(* IEC 61131-3 sources: eCockpitGit/test_project/src/%F%03 Module/%POU%FB_Module/%F%SYS Values/%PRO%SYS_valueUnsigned64, 2 files *)

(* ---- %GETSET%Get.st ---- *)
VAR
END_VAR

(*%!%__DELIMITER__%!%*)
CASE SYS_valueType OF
	EValueType.digital:		SYS_valueUnsigned64	:=		TO_LWORD(SYS_valueDigital);
	EValueType.float32:		SYS_valueUnsigned64	:=		TO_LWORD(SYS_valueFloat32);
	EValueType.enum:			SYS_valueUnsigned64	:=		TO_LWORD(SYS_valueSigned32);

	EValueType.signed32:		SYS_valueUnsigned64	:=		TO_LWORD(SYS_valueSigned32);
	EValueType.unsigned32:	SYS_valueUnsigned64	:=		TO_LWORD(SYS_valueUnsigned32);
	EValueType.signed64:		SYS_valueUnsigned64	:=		TO_LWORD(SYS_valueSigned64);
END_CASE

(* ---- %GETSET%Set.st ---- *)
VAR
END_VAR

(*%!%__DELIMITER__%!%*)
CASE SYS_valueType OF
	EValueType.digital:		SYS_valueDigital		:=		TO_BOOL(SYS_valueUnsigned64);
	EValueType.float32:		SYS_valueFloat32			:=		TO_REAL(SYS_valueUnsigned64);
	EValueType.enum:			SYS_valueSigned32		:=		TO_DINT(SYS_valueUnsigned64);

	EValueType.signed32:		SYS_valueSigned32		:=		TO_DINT(SYS_valueUnsigned64);
	EValueType.unsigned32:	SYS_valueUnsigned32		:=		TO_DWORD(SYS_valueUnsigned64);
	EValueType.signed64:		SYS_valueSigned64		:=		TO_LINT(SYS_valueUnsigned64);
END_CASE
